FUNCTION F_exponential : lreal
VAR_INPUT
	x : LREAL;
END_VAR

F_exponential := exp(x);

END_FUNCTION

(* stored: Version 1.1.0.1, ProductVersion 3.1.4024.12
   POU F_exponential: Id {d871f8f7-3aa5-4062-900b-46dd2ce56fdc}, SpecialFunc None *)
